KUKA KRL data list: dockon_1.dat

&ACCESS RVP1
&REL 164
&COMMENT PICKUP GUN 1
DEFDAT  DOCKON_1
;FOLD EXTERNAL DECLARATIONS;%{PE}%MKUKATPBASIS,%CEXT,%VCOMMON,%P
;FOLD GRIPPERTECH EXT
EXT  H50 (INT  :IN,INT  :IN,INT  :IN,GRP_TYP  :IN )
;ENDFOLD (GRIPPERTECH EXT)
;FOLD SPOTTECH EXT
EXT  USERSPOT (S_COMMAND  :IN,SPOT_TYPE  :IN )
;ENDFOLD (SPOTTECH EXT)
;FOLD BASISTECH EXT;%{PE}%MKUKATPBASIS,%CEXT,%VEXT,%P
EXT  BAS (BAS_COMMAND  :IN,REAL  :IN )
DECL INT SUCCESS
;ENDFOLD (BASISTECH EXT)
;FOLD USER EXT;%{E}%MKUKATPUSER,%CEXT,%VEXT,%P
;Make here your modifications
;ENDFOLD (USER EXT)
;ENDFOLD (EXTERNAL DECLERATIONS)
DECL GRP_TYP GCONT={G_APO #YES,TIME 0.0,CTRL #OFF,DLY 0,DST 0}
DECL GRP_TYP GGDAT={G_APO #NO,TIME 0.0,CTRL #OFF,DLY 0,DST 1}
;*      FDAT Declarations     *

;******************************
;*     E6POS Declarations     *
;******************************

DECL E6POS XP10={X -268.898285,Y 1937.70898,Z 2261.59912,A 150.224899,B 20.9214802,C 81.1931381,S 6,T 59,E1 -735.491699,E2 0.0,E3 0.0,E4 0.0,E5 0.0,E6 0.0}
DECL E6POS XP20={X 1200.62903,Y 1521.23804,Z 2604.01001,A 24.9272804,B 16.2745209,C 74.0746613,S 6,T 27,E1 -1873.25,E2 0.0,E3 0.0,E4 0.0,E5 0.0,E6 0.0}
DECL E6POS XP30={X 89.4970703,Y 846.668274,Z 2110.87402,A -45.796669,B 48.7276192,C 88.0356369,S 6,T 26,E1 -2602.28101,E2 0.0,E3 0.0,E4 0.0,E5 0.0,E6 0.0}
DECL E6POS XP40={X -1098.95203,Y 234.777298,Z 1356.98804,A -91.2462006,B 62.4295502,C 88.7397537,S 6,T 26,E1 -2887.16602,E2 0.0,E3 0.0,E4 0.0,E5 0.0,E6 0.0}
DECL E6POS XP50={X -1235.52698,Y 267.944489,Z 691.163025,A -89.8934402,B 60.7926598,C 90.3862991,S 6,T 26,E1 -2887.16406,E2 0.0,E3 0.0,E4 0.0,E5 0.0,E6 0.0}
DECL E6POS XP60={X -1385.65198,Y 268.574707,Z 690.707581,A -89.8945465,B 60.7910614,C 90.3862991,S 6,T 26,E1 -2887.16211,E2 0.0,E3 0.0,E4 0.0,E5 0.0,E6 0.0}
DECL E6POS XP70={X -1447.02405,Y 268.834198,Z 690.453979,A -89.8933563,B 60.7941017,C 90.3872528,S 6,T 24,E1 -2887.16211,E2 0.0,E3 0.0,E4 0.0,E5 0.0,E6 0.0}
DECL E6POS XP80={X -1267.02698,Y 268.123596,Z 739.39801,A -89.8929367,B 60.793541,C 90.3884506,S 6,T 26,E1 -2887.16406,E2 0.0,E3 0.0,E4 0.0,E5 0.0,E6 0.0}
DECL E6POS XP90={X -1720.43506,Y 93.9415512,Z -744.218323,A 93.5069504,B 77.8008118,C -176.742905,S 6,T 24,E1 -2887.16699,E2 0.0,E3 0.0,E4 0.0,E5 0.0,E6 0.0}
DECL E6POS XP100={X -1472.68103,Y 74.3762131,Z -711.037292,A 124.071701,B 75.2476273,C -145.362396,S 6,T 24,E1 -2887.16895,E2 0.0,E3 0.0,E4 0.0,E5 0.0,E6 0.0}
DECL E6POS XP110={X -958.114685,Y 929.287476,Z 985.58728,A 92.0781479,B 72.5531616,C -179.836502,S 6,T 26,E1 -2887.177,E2 0.0,E3 0.0,E4 0.0,E5 0.0,E6 0.0}

;******************************
;*     FDAT Declarations      *
;******************************

DECL FDAT FP10={TOOL_NO 10,BASE_NO 0,IPO_FRAME #BASE}
DECL FDAT FP20={TOOL_NO 10,BASE_NO 0,IPO_FRAME #BASE}
DECL FDAT FP30={TOOL_NO 10,BASE_NO 0,IPO_FRAME #BASE}
DECL FDAT FP40={TOOL_NO 10,BASE_NO 0,IPO_FRAME #BASE}
DECL FDAT FP50={TOOL_NO 10,BASE_NO 0,IPO_FRAME #BASE}
DECL FDAT FP60={TOOL_NO 10,BASE_NO 0,IPO_FRAME #BASE}
DECL FDAT FP70={TOOL_NO 10,BASE_NO 0,IPO_FRAME #BASE}
DECL FDAT FP80={TOOL_NO 14,BASE_NO 0,IPO_FRAME #BASE}
DECL FDAT FP90={TOOL_NO 1,BASE_NO 0,IPO_FRAME #BASE}
DECL FDAT FP100={TOOL_NO 1,BASE_NO 0,IPO_FRAME #BASE}
DECL FDAT FP110={TOOL_NO 1,BASE_NO 0,IPO_FRAME #BASE}

;******************************
;*  PDAT & LDAT Declarations  *
;******************************

DECL PDAT PH={VEL 100.0,ACC 100.0,APO_DIST 100.0}
DECL LDAT LH={VEL 1.0,ACC 100.0,APO_DIST 100.0,APO_FAC 50.0,ORI_TYP #VAR}

DECL E6POS XP105={X -1401.90906,Y 74.2495728,Z -298.355194,A 148.145004,B 66.4621735,C -119.9972,S 6,T 26,E1 -2887.17505,E2 0.0,E3 0.0,E4 0.0,E5 0.0,E6 0.0}
DECL FDAT Fp105={TOOL_NO 1,BASE_NO 0,IPO_FRAME #BASE,POINT2[] " "}
DECL SPOT_SUGG_T LAST_SPOT={GUN[] "1                       ",RETR_CMD[] "#OPN                    ",CHOISE[] "#FIRST                  ",CLO_TM[] "0                       ",PGNO1[] "1                       ",PRESS1[] "0                       ",PGNO2[] "1                       ",PRESS2[] "0                       ",SPOT_PARAMS[] "SDAT0                   "}
DECL BASIS_SUGG_T LAST_BASIS={POINT1[] "p110                    ",POINT2[] "p110                    ",CP_PARAMS[] "H                       ",PTP_PARAMS[] "H                       ",CONT[] "                        ",CP_VEL[] "2                       ",PTP_VEL[] "100                     "}
DECL E6POS XP81={X -1720.43103,Y 178.551804,Z -744.220276,A 93.51017,B 77.8132935,C -176.7397,S 6,T 26,E1 -2887.16602,E2 0.0,E3 0.0,E4 0.0,E5 0.0,E6 0.0}
DECL FDAT Fp81={TOOL_NO 1,BASE_NO 0,IPO_FRAME #BASE,POINT2[] " "}
ENDDAT
